INTERFACE ITF_Defect EXTENDS __SYSTEM.IQueryInterface

METHOD Ack
END_METHOD

METHOD PUBLIC BuildStringMsg : BOOL
//return false if no error 
VAR_INPUT
	sMsgOut_P               : POINTER TO T_StringBuffer;//return the Telegram message
  sTextOut_P              : POINTER TO T_StringBuffer;//return the ADS console message  
	bConsoleMsg             : BOOL := FALSE;
  
	bShowIstance            : BOOL := FALSE;
  bShowLongClass          : BOOL := FALSE;
  bShowLongError          : BOOL := FALSE;
  bShowRemedMsg           : BOOL := FALSE;
END_VAR
END_METHOD

PROPERTY PUBLIC CanSendAlarmMsg : BOOL
GET
END_GET
END_PROPERTY

PROPERTY PUBLIC CanSendRegisterMsg : BOOL
GET
END_GET
END_PROPERTY

PROPERTY ClassID : STRING(3)
GET
END_GET
END_PROPERTY

PROPERTY ErrorID : STRING(3)
GET
END_GET
END_PROPERTY

PROPERTY FallingEdge : DATE_AND_TIME
GET
END_GET
END_PROPERTY

PROPERTY InstancePath : T_InstancePath
GET
END_GET
END_PROPERTY

METHOD PUBLIC Register : BOOL
VAR_INPUT
	DefectMngr  : REFERENCE TO CL_DefectManager;
  inClassID	  :	STRING(3);
  inErrorID   :	STRING(3);
END_VAR
END_METHOD

PROPERTY RisingEdge : DATE_AND_TIME
GET
END_GET
END_PROPERTY

METHOD Set
VAR_INPUT
  Activate : BOOL;
END_VAR
END_METHOD

METHOD PUBLIC SetOn
VAR_INPUT
END_VAR
END_METHOD

PROPERTY Severity : TcEventSeverity
GET
END_GET
END_PROPERTY

PROPERTY State : E_DefectState
GET
END_GET
END_PROPERTY

END_INTERFACE

(* stored: Version 1.1.0.1, ProductVersion 3.1.4024.12
   Itf ITF_Defect: Id {89b16cf0-c09f-47d5-98b3-546ad3355eb4}
   Method Ack: Id {0fb4237d-1970-47d1-b829-081be3660862}
   Method BuildStringMsg: Id {580b25fe-5b64-4c0e-b775-26b897c582d2}
   Property CanSendAlarmMsg: Id {b74b50b0-24ef-43f2-a79b-586bccdc223d}
   Get Get: Id {f766fca7-db9a-4a42-9baf-68f3cafb7e70}
   Property CanSendRegisterMsg: Id {f46677d4-0f1e-4379-b48f-f4f8136faa61}
   Get Get: Id {e2d9cdba-52b6-4b87-9745-0642f2d63740}
   Property ClassID: Id {78ac3cfb-ecd0-4b8d-afd5-ac03869092ed}
   Get Get: Id {35d24f09-3a95-4116-ac76-77bf31646393}
   Property ErrorID: Id {2055ee96-4912-436f-bbe8-31ccec2804e4}
   Get Get: Id {8b9e9dd6-9f33-4ed8-b309-732df45cd58c}
   Property FallingEdge: Id {86f0caa9-846e-4ade-aa41-e10b149927f4}
   Get Get: Id {fab1dcdc-5d8c-40fe-b596-866f5b2753ce}
   Property InstancePath: Id {6dc0f06c-9792-4a70-af22-59e9811e051e}
   Get Get: Id {86a329a7-002c-460f-ba14-5ef9adc6dbdb}
   Method Register: Id {0c8f1450-e6c4-45ec-9ce7-f94f42898776}
   Property RisingEdge: Id {57bdadbd-21fa-41dd-a3d4-afc667e0ae4e}
   Get Get: Id {0e4552db-98d7-4413-bc07-c6c1450bb1c0}
   Method Set: Id {7882b9e3-a8fb-4fa0-b5bd-b6658a4f19c5}
   Method SetOn: Id {712c1a87-cee9-46ee-ade0-211337a0720c}
   Property Severity: Id {4a5ed5a0-fe89-40ed-a868-4860eafda498}
   Get Get: Id {715f6573-6e24-49e6-ae22-188dbb5c7db3}
   Property State: Id {e9b7f28b-da9f-449b-aaec-ffd6d6f5e638}
   Get Get: Id {ae3bcc9b-957e-49f6-9bed-f6fa7d9acdb2} *)
